FUNCTION_BLOCK RunManual
VAR_INPUT
END_VAR
VAR_OUTPUT
END_VAR
VAR
	wordOut  AT%M* : WORD; //0
	reserved1 AT%M* : ARRAY[1..31] OF WORD;
	wordIn	 AT%M* : WORD; //32
	reserved2 AT%M* : ARRAY[1..8] OF WORD;
	monitorType AT%M* : WORD;//40
	monitorIndex AT%M* : WORD;//41
	commitMode AT%M* : DWORD;//42
	commitSelection AT%M* : DWORD;//44
	commitIndex AT%M* : WORD;//46
	reserved3 AT%M* : ARRAY[1..18] OF WORD;
	dataBlock AT%M* : Block64Words;//64
	monitorBlock AT%M* : Block64Words;//128
	
	monitorDevice : ICommon;
	controlDevice : ICommon;
END_VAR

//monitor
CASE monitorType OF
	eTypeCodes.AXIS:
		monitorDevice := gvl.axisControls[monitorIndex];
	eTypeCodes.CYLINDER:
		monitorDevice := gvl.cylinderControls[monitorIndex];
	eTypeCodes.UNIT:
		monitorDevice := gvl.stations[monitorIndex]^;
END_CASE
monitorBlock := monitorDevice.Monitor();

//

END_FUNCTION_BLOCK

(* stored: Version 1.1.0.1, ProductVersion 3.1.4022.10
   POU RunManual: Id {69f8e896-e3c8-4e08-b157-7fa165a49498}, SpecialFunc None *)
